{attribute 'qualified_only'}
VAR_GLOBAL
	Blink_Slow 	: BOOL	; // Slow blinking bit
	Blink_Fast	: BOOL	; // fast blinking Bit
	
END_VAR
VAR_GLOBAL CONSTANT
	ALWAYS_TRUE		: BOOL := TRUE	; // always true constant
	ALWAYS_FALSE	: BOOL := FALSE	; // ALways false constant 
END_VAR

(* stored: Version 1.1.0.1
   GVL Global_Managed_Variables: Id {13236581-66a9-4c59-a9e4-1f25e6ddbcf6} *)
